Omron Sysmac Studio project Prog_NX-Safety_Att (Sysmac Studio 1.56.0.11, StandardProject)

# Controller new_Controller_0: NJ101-1020 version 1.12
Units and slaves: Node1 : NX-ECC202 (E001); Unit 2 : NX-SID800 (N2); Unit 3 : NX-SOD400 (N3); Unit 4 : NX-ID5442 (N4); Unit 5 : NX-OD5256 (N5); Unit 6 : NX-ILM400 (N6); Unit 7 : NX-EC0112 (N7); Unit 8 : NX-PG0112 (N8); Unit 9 : NX-RS1201 (N9); Power Supply : NJ-Px3001; CPU : NJ101-1020
Axis ESTEIRA, settings changed from default: AxisType=ServoType, UnitsConversion=EnumElement2, UnitsNumerator=8388608, UnitsDenominator=10, MaxVelocity=500, MaxJogVelocity=150, ModuloMAXPosition=10, ModuloMINPosition=0, EncoderTypes=Abs
Axis CONTADOR, settings changed from default: AxisNumber=1, AxisType=ServoType, UnitsConversion=EnumElement5, UnitsNumerator=8388608, UnitsDenominator=360, MaxVelocity=18000, MaxJogVelocity=3000, CountMode=EnumElement2, ModuloMAXPosition=360, ModuloMINPosition=0, EncoderTypes=Abs
Task PrimaryTask (priority 4, period or condition 2000): Program0

VAR_GLOBAL
    Maq_Em_Seguranca : BOOL;  (* at ECAT://node#[1,1]/Maq_CondicaoSegura *)
END_VAR
VAR_GLOBAL CONSTANT
    ESTEIRA : _sAXIS_REF;  (* at MC://_MC_AX[0] *)
    CONTADOR : _sAXIS_REF;  (* at MC://_MC_AX[1] *)
END_VAR
VAR_GLOBAL
    SERVO_EST_ON : BOOL;
    ESTEIRA_HOME_OK : BOOL;
    ZERA_ESTEIRA : BOOL;
    SERVO_CONT_ON : BOOL;
    ZERA_CONTADOR : BOOL;
    CONTADOR_HOME_OK : BOOL;
    START_HORÁRIO_ESTEIRA : BOOL;  (* at ECAT://node#[1,4]/Input Bit 16 bits/Input Bit 00 *)
    ANT_HORÁRIO_ESTEIRA : BOOL;  (* at ECAT://node#[1,4]/Input Bit 16 bits/Input Bit 01 *)
    START_HORARIO_CONTADOR : BOOL;  (* at ECAT://node#[1,4]/Input Bit 16 bits/Input Bit 08 *)
    ANT_HORARIO_CONTADOR : BOOL;  (* at ECAT://node#[1,4]/Input Bit 16 bits/Input Bit 09 *)
END_VAR

(* Program Program0: safety or other program stored in binary form, left out *)

PROGRAM Program0
VAR
    M0 : BOOL;
    BT0 : BOOL;
    POWER_ESTEIRA : MC_Power;
    HOME_ESTEIRA : MC_Home;
    TON_1 : TON;
    POWER_POSICIONADOR : MC_Power;
    HOME_CONTADOR : MC_Home;
    MOVE_ESTEIRA : MC_MoveJog;
    MOVE_CONTADOR : MC_MoveJog;
END_VAR
VAR_EXTERNAL
    Maq_Em_Seguranca : BOOL;
END_VAR
VAR_EXTERNAL CONSTANT
    ESTEIRA : _sAXIS_REF;
END_VAR
VAR_EXTERNAL
    SERVO_EST_ON : BOOL;
    ESTEIRA_HOME_OK : BOOL;
    ZERA_ESTEIRA : BOOL;
END_VAR
VAR_EXTERNAL CONSTANT
    CONTADOR : _sAXIS_REF;
END_VAR
VAR_EXTERNAL
    SERVO_CONT_ON : BOOL;
    ZERA_CONTADOR : BOOL;
    CONTADOR_HOME_OK : BOOL;
    START_HORÁRIO_ESTEIRA : BOOL;
    ANT_HORÁRIO_ESTEIRA : BOOL;
    START_HORARIO_CONTADOR : BOOL;
    ANT_HORARIO_CONTADOR : BOOL;
END_VAR

(* Section Section0: ladder, written here as Structured Text *)

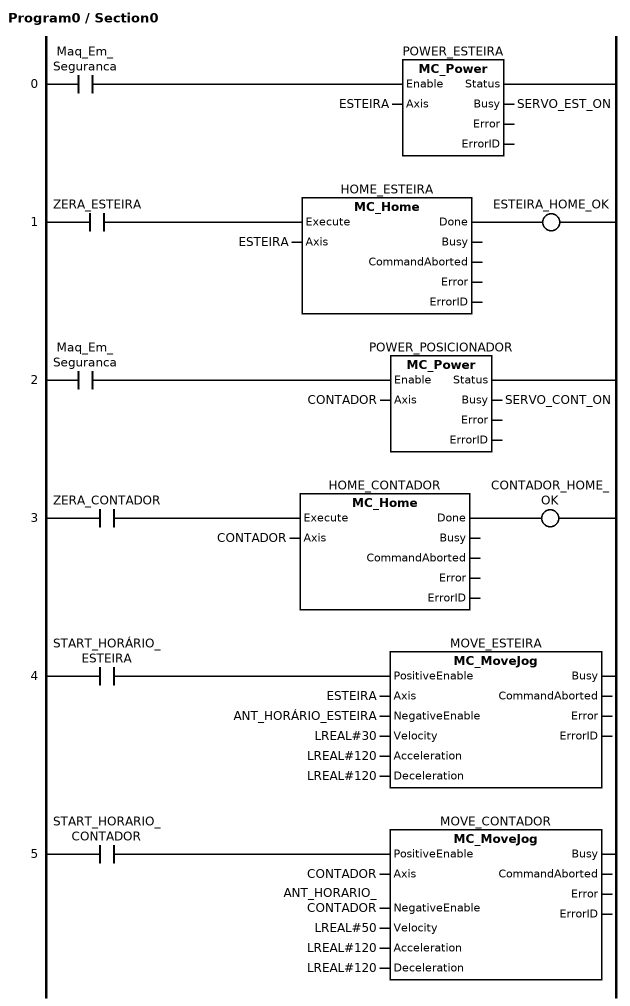
(* Rung 0 *)
POWER_ESTEIRA(Enable := Maq_Em_Seguranca, Axis := ESTEIRA, Busy => SERVO_EST_ON);
(* Rung 1 *)
HOME_ESTEIRA(Execute := ZERA_ESTEIRA, Axis := ESTEIRA);
ESTEIRA_HOME_OK := HOME_ESTEIRA.Done;
(* Rung 2 *)
POWER_POSICIONADOR(Enable := Maq_Em_Seguranca, Axis := CONTADOR, Busy => SERVO_CONT_ON);
(* Rung 3 *)
HOME_CONTADOR(Execute := ZERA_CONTADOR, Axis := CONTADOR);
CONTADOR_HOME_OK := HOME_CONTADOR.Done;
(* Rung 4 *)
MOVE_ESTEIRA(PositiveEnable := START_HORÁRIO_ESTEIRA, Axis := ESTEIRA, NegativeEnable := ANT_HORÁRIO_ESTEIRA, Velocity := LREAL#30, Acceleration := LREAL#120, Deceleration := LREAL#120);
(* Rung 5 *)
MOVE_CONTADOR(PositiveEnable := START_HORARIO_CONTADOR, Axis := CONTADOR, NegativeEnable := ANT_HORARIO_CONTADOR, Velocity := LREAL#50, Acceleration := LREAL#120, Deceleration := LREAL#120);
END_PROGRAM